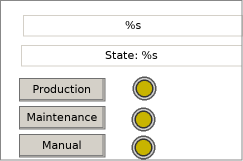
VISUALIZATION V_Module  // 243x161
VAR_IN_OUT
	HMI : ST_PackMLBaseModule_HMI;
END_VAR
    Textfield (23,15 220x21), "%s", text variable: HMI.Config.Name
    Textfield (21,45 221x21), "State: %s", text variable: HMI.Status.State
    Button (19,78 86x23), "Production"
        OnMouseClick: execute { HMI.Command.Mode := E_PMLUnitMode.ePMLUnitMode_Production; }
    Button (19,106 86x23), "Maintenance"
        OnMouseClick: execute { HMI.Command.Mode := E_PMLUnitMode.ePMLUnitMode_Maintenance; }
    Button (19,134 86x23), "Manual"
        OnMouseClick: execute { HMI.Command.Mode := E_PMLUnitMode.ePMLUnitMode_Manual; }
    Lamp1 (131,75 27x27), variable: HMI.Status.Mode = E_PMLUnitMode.ePMLUnitMode_Production, style: Lamp-Lamp1-Yellow
    Lamp1 (130,106 27x27), variable: HMI.Status.Mode = E_PMLUnitMode.ePMLUnitMode_Maintenance, style: Lamp-Lamp1-Yellow
    Lamp1 (130,134 27x27), variable: HMI.Status.Mode = E_PMLUnitMode.ePMLUnitMode_Manual, style: Lamp-Lamp1-Yellow
END_VISUALIZATION

(* stored: Version 1.1.0.1
   Visu V_Module: Id {ab5ca517-81c1-49dd-92aa-b6c97677d45a} *)
